{attribute 'qualified_only'}
{attribute 'strict'}
TYPE E_PFH_InitState : // Parameter file handler (PFH) init state
(
	InitialState,
	OpenFile,
	CreateFile,
	WriteRecord,
	WriteRecordBusy,
	ReadRecord,
	ParseRecord,
	CloseFile,
	Done,
	Error
);
END_TYPE

(* stored: Version 1.1.0.1, ProductVersion 3.1.4024.11
   DUT E_PFH_InitState: Id {c51eac8f-cae4-067a-33c0-c0715d3aafd1} *)
